(* PLC project Tc3_EventLogger.EqualsToEventClass Demo, tc3-libraries-kb TwinCAT 3.1 *)
(* stored: creationDateTime 2026-05-11T01:00:00, modificationDateTime 2026-05-11T01:00:00 *)

PROGRAM P_Demo_EqualsToEventClass
  VAR
    fbAlarm : FB_TcAlarm;  (* alarm 实例 *)
    guidExpected : GUID;  (* 要匹配的事件类 GUID *)
    bMatch : BOOL;  (* 比较结果 *)
  END_VAR

// =============================================================================
// 场景：判断当前 alarm 是否属于「安全报警」类
// 价值：一次调用即可分流
// 验证：登录后让 fbAlarm.Create 用某 GUID，再写 guidExpected 为相同 GUID → bMatch=TRUE；改 guidExpected 任一字节 → FALSE
// 验证步骤：
//   1. 右键 PLC 项目 → Import PLCopenXML → 选本文件
//   2. 引用 Tc3_EventLogger（System → References → Add library）
//   3. 编译 → 登录 → 运行；按 verify 注释里给出的在线写值操作
// =============================================================================

// 调用者已经持有 alarm 实例，判断它是否属于 guidExpected 这个事件类
bMatch := fbAlarm.EqualsToEventClass(eventClass := guidExpected);
END_PROGRAM
